# EPICS substitutions: utcaApp/Db/bpm_data.substitutions
file db/bpm_data.template {
    pattern {ADC, ADDR}
    {"A", 0}
    {"B", 1}
    {"C", 2}
    {"D", 3}
}
